// TIA Portal V19 export
FUNCTION "FC_FW_Auftrag_Step3_NB" : Void   // FC183, LAD
TITLE = Schritt CM03 -> CM04
{ S7_Optimized_Access := 'TRUE' }
// Ältesten Warenträger in CM03 suchen und nach CM04 transportieren
// stored: AutoNumber false, SetENOAutomatically false
   VAR_INPUT
      Frg_Schritt : Bool;
   END_VAR
   VAR_OUTPUT
      nextStep : Bool;
      startStep : Bool;
      parkStep : Bool;
   END_VAR
   VAR_IN_OUT
      Quelle : Int;
      Ziel : Int;
      Positionen : Array[1..30] of "UDT_Auftrag_Pos";
   END_VAR
   VAR_TEMP
      Sperre_Kurz_li : Bool;
      Sperre_Kurz_re : Bool;
      Sperre_Lang : Bool;
      Vorzug : Bool;
      Befehl_ok : Bool;
      tmpQuelle : Int;
      Oldest : Real;
   END_VAR
   VAR CONSTANT
      Wt_Cmd_Aetzen : Int := 1;
   END_VAR
BEGIN

REGION Network 1 (SCL)
   IF (#Quelle <> 0) AND (#Ziel <> 0) THEN
       #nextStep := #Positionen[#Quelle].Sperre;
       #startStep := NOT #nextStep;
       #Quelle := 0;
       #Ziel := 0;
       RETURN;
   END_IF;

   #Quelle := 0;
   #Ziel := 0;
   #nextStep := FALSE;
   #startStep := FALSE;

   IF NOT #Frg_Schritt THEN
       #nextStep := TRUE;
       RETURN;
   END_IF;
END_REGION

REGION Network 2 (SCL): Positionen sperren
   //Groß links nicht möglich
   #Positionen[9].CheckSperre := #Positionen[21].Sperre OR (#Positionen[9].Wt_Cmd = #Wt_Cmd_Aetzen);

   //Groß rechts nicht möglich
   #Positionen[10].CheckSperre := #Positionen[22].Sperre OR (#Positionen[10].Wt_Cmd = #Wt_Cmd_Aetzen);

   //kein Platz für Kurz links in CM04
   #Sperre_Kurz_li := #Positionen[19].Sperre AND #Positionen[23].Sperre;

   //kein Platz für Kurz rechts in CM04
   #Sperre_Kurz_re := #Positionen[20].Sperre AND #Positionen[24].Sperre;

   //kein Platz für Lang in CM04
   #Sperre_Lang := (#Positionen[19].Sperre OR #Positionen[20].Sperre) AND (#Positionen[23].Sperre OR #Positionen[24].Sperre);

   //Lang in P7 oder
   //kein Platz auf rechter Seite
   //-> P8 sperren
   #Positionen[8].CheckSperre := #Sperre_Kurz_re OR (#Positionen[7].Wt_Typ = "WT_Typ_LS") OR (#Positionen[8].Wt_Cmd = #Wt_Cmd_Aetzen);

   //Lang in P7 und kein Platz für Lang oder
   //kein Platz auf linker Seite
   //-> P7 sperren
   #Positionen[7].CheckSperre := #Sperre_Kurz_li OR ((#Positionen[7].Wt_Typ = "WT_Typ_LS") AND #Sperre_Lang) OR (#Positionen[7].Wt_Cmd = #Wt_Cmd_Aetzen);

   //Lang in P11 oder
   //kein Platz auf rechter Seite
   //-> P12 sperren
   #Positionen[12].CheckSperre := #Sperre_Kurz_re OR (#Positionen[11].Wt_Typ = "WT_Typ_LS") OR (#Positionen[12].Wt_Cmd = #Wt_Cmd_Aetzen);

   //Lang in P11 und kein Platz für Lang oder
   //kein Platz auf linker Seite
   //-> P11 sperren
   #Positionen[11].CheckSperre := #Sperre_Kurz_li OR ((#Positionen[11].Wt_Typ = "WT_Typ_LS") AND #Sperre_Lang) OR (#Positionen[11].Wt_Cmd = #Wt_Cmd_Aetzen);
END_REGION

REGION Network 3 (SCL): Ältesten WT suchen
   //
   #Oldest := 0;
   #tmpQuelle := 0;

   //CM03
   "FC_FW_Auftrag_Suche"(Pos1 := 7,
                         Pos2 := 12,
                         Positionen := #Positionen,
                         Quelle := #tmpQuelle,
                         Oldest := #Oldest);
END_REGION

REGION Network 4 (SCL): Auswertung
   IF #tmpQuelle = 0 THEN
       //kein WT
       #nextStep := TRUE;
       RETURN;
   END_IF;

   IF NOT #Positionen[#tmpQuelle].Fertig THEN
       #parkStep := TRUE;
       RETURN;
   END_IF;

   IF (#tmpQuelle = 9) THEN
       //Gross links
       IF NOT #Positionen[21].Sperre THEN
           "FC_FW_Auftrag_Befehl"(inQuelle := #tmpQuelle,
                                  inZiel := 21,
                                  Befehl_ok => #Befehl_ok,
                                  outQuelle => #Quelle,
                                  outZiel => #Ziel);

           #nextStep := NOT #Befehl_ok;
       ELSE
           #nextStep := TRUE;
       END_IF;
       RETURN;
   END_IF;

   IF (#tmpQuelle = 10) THEN
       //Gross rechts
       IF NOT #Positionen[22].Sperre THEN
           "FC_FW_Auftrag_Befehl"(inQuelle := #tmpQuelle,
                                  inZiel := 22,
                                  Befehl_ok => #Befehl_ok,
                                  outQuelle => #Quelle,
                                  outZiel => #Ziel);

           #nextStep := NOT #Befehl_ok;
       ELSE
           #nextStep := TRUE;
       END_IF;
       RETURN;
   END_IF;

   IF (#Positionen[#tmpQuelle].Wt_Typ = "WT_Typ_LS") AND ((#tmpQuelle = 7) OR (#tmpQuelle = 11)) THEN
       //Lang
       IF NOT #Positionen[19].Sperre AND NOT #Positionen[20].Sperre THEN
           "FC_FW_Auftrag_Befehl"(inQuelle := #tmpQuelle,
                                  inZiel := 19,
                                  Befehl_ok => #Befehl_ok,
                                  outQuelle => #Quelle,
                                  outZiel => #Ziel);

           #nextStep := NOT #Befehl_ok;
       ELSIF NOT #Positionen[23].Sperre AND NOT #Positionen[24].Sperre THEN
           "FC_FW_Auftrag_Befehl"(inQuelle := #tmpQuelle,
                                  inZiel := 23,
                                  Befehl_ok => #Befehl_ok,
                                  outQuelle => #Quelle,
                                  outZiel => #Ziel);

           #nextStep := NOT #Befehl_ok;
       ELSE
           #nextStep := TRUE;
       END_IF;
       RETURN;
   END_IF;

   IF (#tmpQuelle = 7) OR (#tmpQuelle = 11) THEN
       //Kurz links
       #Vorzug := NOT #Positionen[19].Sperre AND NOT #Positionen[20].Sperre AND NOT #Positionen[23].Sperre AND #Positionen[24].Sperre;

       IF NOT #Positionen[19].Sperre AND NOT #Vorzug THEN
           "FC_FW_Auftrag_Befehl"(inQuelle := #tmpQuelle,
                                  inZiel := 19,
                                  Befehl_ok => #Befehl_ok,
                                  outQuelle => #Quelle,
                                  outZiel => #Ziel);

           #nextStep := NOT #Befehl_ok;
       ELSIF NOT #Positionen[23].Sperre THEN
           "FC_FW_Auftrag_Befehl"(inQuelle := #tmpQuelle,
                                  inZiel := 23,
                                  Befehl_ok => #Befehl_ok,
                                  outQuelle => #Quelle,
                                  outZiel => #Ziel);

           #nextStep := NOT #Befehl_ok;
       ELSE
           #nextStep := TRUE;
       END_IF;
       RETURN;
   END_IF;

   IF (#tmpQuelle = 8) OR (#tmpQuelle = 12) THEN
       //Kurz rechts
       #Vorzug := NOT #Positionen[19].Sperre AND NOT #Positionen[20].Sperre AND #Positionen[23].Sperre AND NOT #Positionen[24].Sperre;

       IF NOT #Positionen[20].Sperre AND NOT #Vorzug THEN
           "FC_FW_Auftrag_Befehl"(inQuelle := #tmpQuelle,
                                  inZiel := 20,
                                  Befehl_ok => #Befehl_ok,
                                  outQuelle => #Quelle,
                                  outZiel => #Ziel);

           #nextStep := NOT #Befehl_ok;
       ELSIF NOT #Positionen[24].Sperre THEN
           "FC_FW_Auftrag_Befehl"(inQuelle := #tmpQuelle,
                                  inZiel := 24,
                                  Befehl_ok => #Befehl_ok,
                                  outQuelle => #Quelle,
                                  outZiel => #Ziel);

           #nextStep := NOT #Befehl_ok;
       ELSE
           #nextStep := TRUE;
       END_IF;
       RETURN;
   END_IF;

   //?
   #nextStep := TRUE;
END_REGION
END_FUNCTION
